INTERFACE ITF_EventHandler

METHOD PUBLIC CmdAddFault : BOOL
VAR_IN_OUT
	stFault : UDT_Fault ; // actuive fault structure input
END_VAR
END_METHOD

METHOD PUBLIC CmdReset : BOOL
VAR_INPUT
END_VAR
END_METHOD

END_INTERFACE

(* stored: Version 1.1.0.1, ProductVersion 3.1.4024.9
   Itf ITF_EventHandler: Id {e0ad6bc5-60ea-49db-af8f-6d978affa684}
   Method CmdAddFault: Id {7c67df34-80af-4fe4-8ff2-cc9ec23a1c1e}
   Method CmdReset: Id {87c6c083-318a-44e4-b567-19b90f95408e} *)
